FUNCTION_BLOCK FB_PistonExtruderControl EXTENDS FB_ExtruderControl

VAR
	eSubType				: E_ExtruderType;
	pFbPistonExtruderRef	: POINTER TO FB_PistonExtruderRef;
	nStateSdo 				: USINT;
	nNextStateSdo			: USINT;
	fbSdoWrite				: FB_SDO_WRITE;
	bSendDistancePending	: BOOL;
	bSendUnlockOffsetPending: BOOL;
	fbList					: FB_LinkedListCtrl;
	hList					: T_HLINKEDLIST;
	aListNodes				: ARRAY[0..6] OF T_LinkedListEntry;
	nListValue				: PVOID;
	
	bLock					: BOOL;
	nLockOffset				: DINT;
	bUnlock					: BOOL;
	nUnlockOffset			: DINT;
	bMovePlunger			: BOOL;
	nMovePos				: DINT;
	nMoveDistance			: DINT;
	nMoveFeed				: DINT;
	bExtrude				: BOOL;
	
	nCompDistanceTemp		: DINT;
	nRelaxDistanceTemp		: DINT;
	nRelaxFeedTemp			: DINT;
	nDistanceTemp			: DINT;
	nFeedTemp				: DINT;
	
	nStateAction			: USINT;
	
	timer					: TON;
	
	bStop					: BOOL;

END_VAR

VAR CONSTANT
	cMaxPosPiston	 		: DINT := 65000;//µm
	cMaxPosSyringe			: DINT := 87000;//µm
	cMaxFeedPiston			: DINT := 3000;//µm/s
	cMaxFeedSyringe			: DINT := 12000;//µm/s
END_VAR

IF pFbExtruderRef = 0 THEN
	RETURN;
END_IF

pFbPistonExtruderRef := pFbExtruderRef;

IF nStateSdo = 0 THEN //nächsten Eintrag aus Liste holen
	fbList.A_GetHead(hList:= hList,getValue=> nListValue);
	IF fbList.bOk THEN
		{IF  hasvalue (RegisterSize, '32')}
		nStateSdo := UDINT_TO_USINT(nListValue);
		{ELSE}
		nStateSdo := ULINT_TO_USINT(nListValue);
		{END_IF}		
		fbList.A_RemoveHeadValue(hList:= hList);
	END_IF
END_IF

IF nStateSdo = 1 THEN	//Feed
	fbSdoWrite(sADSNetID:= pFbPistonExtruderRef^.pMultiZRef^.P_sAdsNetId, nPortNr:= pFbPistonExtruderRef^.pMultiZRef^.P_nAdsPort, 
				nIndex:= cExtruderFeed.nIndex, nSubIndex:= pFbPistonExtruderRef^.nChannel, nDataLength:= cExtruderFeed.nLength,
				nData:= pFbPistonExtruderRef^.P_nFeedCalc, bExecute:= TRUE); 
	
ELSIF nStateSdo = 2 THEN //CompressFeed
	fbSdoWrite(sADSNetID:= pFbPistonExtruderRef^.pMultiZRef^.P_sAdsNetId, nPortNr:= pFbPistonExtruderRef^.pMultiZRef^.P_nAdsPort, 
				nIndex:= cExtruderCompressFeed.nIndex, nSubIndex:= pFbPistonExtruderRef^.nChannel, nDataLength:= cExtruderCompressFeed.nLength,
				nData:= pFbPistonExtruderRef^.P_nCompFeedCalc, bExecute:= TRUE); 
	
ELSIF nStateSdo = 3 THEN //RelaxFeed
	fbSdoWrite(sADSNetID:= pFbPistonExtruderRef^.pMultiZRef^.P_sAdsNetId, nPortNr:= pFbPistonExtruderRef^.pMultiZRef^.P_nAdsPort, 
				nIndex:= cExtruderRelaxFeed.nIndex, nSubIndex:= pFbPistonExtruderRef^.nChannel, nDataLength:= cExtruderRelaxFeed.nLength,
				nData:= pFbPistonExtruderRef^.P_nRelaxFeedCalc, bExecute:= TRUE); 
	
ELSIF nStateSdo = 4 THEN //Distance
	fbSdoWrite(sADSNetID:= pFbPistonExtruderRef^.pMultiZRef^.P_sAdsNetId, nPortNr:= pFbPistonExtruderRef^.pMultiZRef^.P_nAdsPort, 
				nIndex:= cExtruderDistance.nIndex, nSubIndex:= pFbPistonExtruderRef^.nChannel, nDataLength:= cExtruderDistance.nLength,
				nData:= pFbPistonExtruderRef^.P_nDistanceCalc, bExecute:= TRUE);
	
ELSIF nStateSdo = 5 THEN //CompressDistance
	fbSdoWrite(sADSNetID:= pFbPistonExtruderRef^.pMultiZRef^.P_sAdsNetId, nPortNr:= pFbPistonExtruderRef^.pMultiZRef^.P_nAdsPort, 
				nIndex:= cExtruderCompressDistance.nIndex, nSubIndex:= pFbPistonExtruderRef^.nChannel, nDataLength:= cExtruderCompressDistance.nLength,
				nData:= pFbPistonExtruderRef^.P_nCompDistanceCalc, bExecute:= TRUE);

ELSIF nStateSdo = 6 THEN //RelaxDistance
	fbSdoWrite(sADSNetID:= pFbPistonExtruderRef^.pMultiZRef^.P_sAdsNetId, nPortNr:= pFbPistonExtruderRef^.pMultiZRef^.P_nAdsPort, 
				nIndex:= cExtruderRelaxDistance.nIndex, nSubIndex:= pFbPistonExtruderRef^.nChannel, nDataLength:= cExtruderRelaxDistance.nLength,
				nData:= pFbPistonExtruderRef^.P_nRelaxDistanceCalc, bExecute:= TRUE);
				
ELSIF nStateSdo = 7 THEN //UnlockOffset
	fbSdoWrite(sADSNetID:= pFbPistonExtruderRef^.pMultiZRef^.P_sAdsNetId, nPortNr:= pFbPistonExtruderRef^.pMultiZRef^.P_nAdsPort, 
				nIndex:= cExtruderUnlockOffset.nIndex, nSubIndex:= pFbPistonExtruderRef^.nChannel, nDataLength:= cExtruderUnlockOffset.nLength,
				nData:= pFbPistonExtruderRef^.P_nUnlockOffsetCalc, bExecute:= TRUE);				
END_IF

IF NOT fbSdoWrite.bBusy THEN
	IF fbSdoWrite.bError THEN
		bError := TRUE;
		nErrorId := fbSdoWrite.nAdsErrorId;		
	END_IF
	fbSdoWrite(bExecute:= FALSE);
	IF nStateSdo = 4 THEN
		bSendDistancePending := FALSE;
	ELSIF nStateSdo = 7 THEN
		bSendUnlockOffsetPending := FALSE;
	END_IF
	nStateSdo := 0;
END_IF


IF bLock THEN
	A_Lock();
ELSIF bUnlock THEN
	A_Unlock();
ELSIF bMovePlunger THEN
	A_MovePlunger();
ELSIF bExtrude THEN
	A_Extrude();
END_IF

IF nStateAction >= 80 THEN
	IF nStateAction >= 99 THEN
		bError := TRUE;
	END_IF
	bLock := bUnlock := bMovePlunger := bExtrude := FALSE;
	nStateAction := 0;
END_IF

bBusy := bLock OR bUnlock OR bMovePlunger OR bExtrude;

ACTION A_Extrude:
CASE nStateAction OF
	0:	//warten, bis Distance gesendet
		IF NOT bSendDistancePending THEN
			pFbPistonExtruderRef^.pToolCtrl^.0 := TRUE;
			nStateAction := 1;				
		END_IF
		
	1:	//Timeout für active
		timer(IN:=TRUE,PT:=T#1S);
		IF pFbPistonExtruderRef^.P_bIsActive THEN
			timer(IN:=FALSE);
			nStateAction := 2;
		ELSE
			IF timer.Q THEN
				timer(IN:=FALSE);
				nErrorId := E_ErrorIdMultiZ.ERRORID_TimeoutExtrude;
				pFbPistonExtruderRef^.pToolCtrl^ := 0;
				nStateAction := 99;
			END_IF
		END_IF
		
	2:	//warten, bis Extrude fertig
		IF NOT pFbPistonExtruderRef^.P_bIsActive OR bStop THEN
			bStop := FALSE;
			pFbPistonExtruderRef^.pToolCtrl^.0 := FALSE;
			nStateAction := 80;
		END_IF
	
END_CASE
END_ACTION

ACTION A_Lock:
CASE nStateAction OF
	0:	//Wartezyklus
		IF pFbPistonExtruderRef^.P_bIsActive THEN
			nStateAction := 99;
		ELSE
			nStateAction := 1;
		END_IF
	1:	//Locking starten
		pFbPistonExtruderRef^.pToolCtrl^.0 := TRUE;
		pFbPistonExtruderRef^.pToolCtrl^.2 := TRUE;
		//Timeout für active
		timer(IN:=TRUE,PT:=T#1S);
		IF pFbPistonExtruderRef^.P_bIsActive THEN
			pFbPistonExtruderRef^.pToolCtrl^.0 := FALSE;
			timer(IN:=FALSE);
			nStateAction := 2;
		ELSE
			IF timer.Q THEN
				timer(IN:=FALSE);
				nErrorId := E_ErrorIdMultiZ.ERRORID_TimeoutLock;
				nStateAction := 99;
			END_IF
		END_IF
		
	2:	//waiting for "ready state"
		timer(IN:=TRUE,PT:=T#25S);
		IF NOT pFbPistonExtruderRef^.P_bIsActive THEN
			timer(IN:=FALSE);
			IF nLockOffset > 0 AND NOT pFbPistonExtruderRef^.pToolCtrl^.1 THEN
				nStateAction := 3;
			ELSE
				nStateAction := 80;
			END_IF
			pFbPistonExtruderRef^.pToolCtrl^ := 0;
		ELSE
			IF timer.Q THEN
				timer(IN:=FALSE);
				nErrorId := E_ErrorIdMultiZ.ERRORID_TimeoutLock;
				nStateAction := 99;
			END_IF
		END_IF
		
	3:	//auf Offset fahren
		//aktuelle CompDistance, RelaxDistance, Feed, Distance sichern
		nCompDistanceTemp := pFbPistonExtruderRef^.P_nCompDistanceOrgin;
		nRelaxDistanceTemp := pFbPistonExtruderRef^.P_nRelaxDistanceOrgin;
		nFeedTemp := pFbPistonExtruderRef^.P_nFeedOrgin;
		nDistanceTemp := pFbPistonExtruderRef^.P_nDistanceOrgin;
		
		//CompDist + RelaxDist auf 0 setzen
		M_SetCompDistance(0);
		M_SetRelaxDistance(0);
		nMoveFeed := M_SetFeedToMax();
		M_SetDistance(nLockOffset); //Distance auf Offset setzen
		nStateAction := 4;
		
	4:	//warten bis Distance gesendet (andere werden vorher gesendet)
		IF NOT bSendDistancePending THEN
			pFbPistonExtruderRef^.pToolCtrl^.0 := TRUE;
			timer(IN:=FALSE);
			nStateAction := 5;
		END_IF
		
	5:	//waiting for "active state"
		timer(IN:=TRUE,PT:=T#1S);
		IF pFbPistonExtruderRef^.P_bIsActive THEN
			timer(IN:=FALSE);
			//timeout berechnen
			timer.PT := REAL_TO_TIME((DINT_TO_REAL(nLockOffset) / DINT_TO_REAL(nMoveFeed))*10000.0 + 3000.0);
			nStateAction := 6;
		ELSE
			IF timer.Q THEN
				timer(IN:=FALSE);
				nErrorId := E_ErrorIdMultiZ.ERRORID_TimeoutLock;
				nStateAction := 7;
			END_IF
		END_IF
		
	6:	//waiting for "ready state"
		timer(IN:=TRUE);
		IF NOT pFbPistonExtruderRef^.P_bIsActive THEN
			timer(IN:=FALSE);
			pFbPistonExtruderRef^.pToolCtrl^ := 0;
			nStateAction := 7;
		ELSE
			IF timer.Q THEN
				timer(IN:=FALSE);
				nErrorId := E_ErrorIdMultiZ.ERRORID_TimeoutLock;
				nStateAction := 7;
			END_IF
		END_IF
		
	7:	//gesicherte Parameter zurückschreiben
		M_SetCompDistance(nCompDistanceTemp);
		M_SetRelaxDistance(nRelaxDistanceTemp);
		M_SetFeed(nFeedTemp);
		M_SetDistance(nDistanceTemp);
		nStateAction := 8;

	8:	//warten bis Distance gesendet (andere werden vorher gesendet)
		IF NOT bSendDistancePending THEN
			IF nErrorId > 0 THEN
				nStateAction := 99;
			ELSE
				nStateAction := 80;
			END_IF
		END_IF		

END_CASE

IF nStateAction = 99 THEN
	pFbPistonExtruderRef^.pToolCtrl^ := 0;
END_IF
END_ACTION

ACTION A_MovePlunger:
//Ähnlich wie Extrude impl.
//vorher aktuelle Position von Zielposition abziehen
//CompDist und RelaxDist auf 0 setzen
CASE nStateAction OF
	0:	//aktuelle CompDistance, RelaxDistance, Feed, Distance sichern
		nCompDistanceTemp := pFbPistonExtruderRef^.P_nCompDistanceOrgin;
		nRelaxDistanceTemp := pFbPistonExtruderRef^.P_nRelaxDistanceOrgin;
		nRelaxFeedTemp := pFbPistonExtruderRef^.P_nRelaxFeedOrgin;
		nFeedTemp := pFbPistonExtruderRef^.P_nFeedOrgin;
		nDistanceTemp := pFbPistonExtruderRef^.P_nDistanceOrgin;
		
		nStateAction := 1;

		M_SetCompDistance(0);
		IF nMovePos > pFbPistonExtruderRef^.P_nCurrentPos THEN
			M_SetRelaxDistance(0);
			nMoveFeed := M_SetFeedToMax();
			nMoveDistance := nMovePos - pFbPistonExtruderRef^.P_nCurrentPos; 
			M_SetDistance(nMoveDistance);
		ELSIF nMovePos < pFbPistonExtruderRef^.P_nCurrentPos THEN
			nMoveDistance := pFbPistonExtruderRef^.P_nCurrentPos - nMovePos;
			M_SetRelaxDistance(nMoveDistance);
			nMoveFeed := M_SetRelaxFeedToMax();
			M_SetFeedToMax();
			M_SetDistance(1);
		ELSE
			nStateAction := 80;
			RETURN;
		END_IF
		
	1:	//warten bis Distance gesendet (andere werden vorher gesendet)
		IF NOT bSendDistancePending THEN
			pFbPistonExtruderRef^.pToolCtrl^.0 := TRUE;
			nStateAction := 2;
		END_IF
		
	2:	//waiting for "active state"
		timer(IN:=TRUE,PT:=T#1S);
		IF pFbPistonExtruderRef^.P_bIsActive THEN
			timer(IN:=FALSE);
			//timeout berechnen
			timer.PT := REAL_TO_TIME((DINT_TO_REAL(nMoveDistance) / DINT_TO_REAL(nMoveFeed))*10000.0 + 3000.0);
			nStateAction := 3;
		ELSE
			IF timer.Q THEN
				timer(IN:=FALSE);
				nErrorId := E_ErrorIdMultiZ.ERRORID_TimeoutMovePlunger;
				nStateAction := 4;
			END_IF
		END_IF	
		
	3:	//warten, bis Extrude fertig
		timer(IN:=TRUE);
		IF NOT pFbPistonExtruderRef^.P_bIsActive THEN
			timer(IN:=FALSE);
			pFbPistonExtruderRef^.pToolCtrl^ := 0;
			nStateAction := 4;
		ELSE
			IF timer.Q THEN
				timer(IN:=FALSE);
				nErrorId := E_ErrorIdMultiZ.ERRORID_TimeoutMovePlunger;
				nStateAction := 4;
			END_IF
		END_IF
		
	4:	//gesicherte Parameter zurückschreiben
		M_SetCompDistance(nCompDistanceTemp);
		M_SetRelaxDistance(nRelaxDistanceTemp);
		M_SetRelaxFeed(nRelaxFeedTemp);
		M_SetFeed(nFeedTemp);
		M_SetDistance(nDistanceTemp);
		nStateAction := 5;
		
	5:	//warten bis Distance gesendet (andere werden vorher gesendet)
		IF NOT bSendDistancePending THEN
			IF nErrorId > 0 THEN
				nStateAction := 99;
			ELSE
				nStateAction := 80;	
			END_IF
		END_IF			
END_CASE

IF nStateAction = 99 THEN
	pFbPistonExtruderRef^.pToolCtrl^ := 0;
END_IF
END_ACTION

ACTION A_Unlock:
CASE nStateAction OF
	0:	//warten bis nUnlockOffset übertragen
		IF NOT bSendUnlockOffsetPending THEN
			nStateAction := 1;
		END_IF
		
	1:	//UnLocking starten
		pFbPistonExtruderRef^.pToolCtrl^.0 := TRUE;
		pFbPistonExtruderRef^.pToolCtrl^.2 := TRUE;
		//Timeout für active
		timer(IN:=TRUE,PT:=T#1S);
		IF pFbPistonExtruderRef^.P_bIsActive THEN
			pFbPistonExtruderRef^.pToolCtrl^.0 := FALSE;
			timer(IN:=FALSE);
			nStateAction := 2;
		ELSE
			IF timer.Q THEN
				timer(IN:=FALSE);
				nErrorId := E_ErrorIdMultiZ.ERRORID_TimeoutUnLock;
				nStateAction := 99;
			END_IF
		END_IF
		
	2:	//warten, bis UnLocking ready
		timer(IN:=TRUE,PT:=T#70S);
		IF NOT pFbPistonExtruderRef^.P_bIsActive THEN
			timer(IN:=FALSE);
			pFbPistonExtruderRef^.pToolCtrl^ := 0;
			nStateAction := 80;
		ELSE
			IF timer.Q THEN
				timer(IN:=FALSE);
				nErrorId := E_ErrorIdMultiZ.ERRORID_TimeoutUnLock;
				nStateAction := 99;
			END_IF
		END_IF
END_CASE

IF nStateAction = 99 THEN
	pFbPistonExtruderRef^.pToolCtrl^ := 0;
END_IF
END_ACTION

METHOD FB_init : BOOL
VAR_INPUT
	bInitRetains : BOOL; // if TRUE, the retain variables are initialized (warm start / cold start)
	bInCopyCode : BOOL;  // if TRUE, the instance afterwards gets moved into the copy code (online change)
END_VAR
F_CreateLinkedListHnd(ADR(aListNodes ), SIZEOF(aListNodes ), hList);
END_METHOD

METHOD PRIVATE M_Add
VAR_INPUT
	nValue : UDINT;
END_VAR
VAR
	pPosPtr	: POINTER TO T_LinkedListEntry := 0;
END_VAR
//Checken, ob Eintrag schon vorhanden
fbList.A_GetHead(hList:= hList,getValue=> nListValue, getPosPtr=> pPosPtr);
IF fbList.bOk THEN
	IF nValue = nListValue THEN	//Eintrag schon vorhanden
		RETURN;		
	ELSE //Eintrag nicht vorhanden -> weitersuchen
		REPEAT
			fbList.A_GetNext(hList:= hList,getValue=> nListValue, putPosPtr:= pPosPtr, getPosPtr=> pPosPtr);
			IF fbList.bOk THEN
				IF nValue = nListValue THEN	//Eintrag schon vorhanden
					RETURN;
				END_IF
			END_IF
		UNTIL NOT fbList.bOk
		END_REPEAT
	END_IF
END_IF

fbList.A_AddTailValue(hList:= hList, putValue:= nValue);
END_METHOD

METHOD M_HardStop
VAR_INPUT
END_VAR
IF pFbPistonExtruderRef^.P_bIsActive THEN
	pFbPistonExtruderRef^.pToolCtrl^ := 2;
END_IF
END_METHOD

METHOD M_Init
VAR_INPUT
END_VAR

VAR
	i : USINT;
END_VAR
//Alle Parameter übertragen
FOR i := 1 TO 7 BY 1 DO
	M_Add(i);
END_FOR
END_METHOD

METHOD M_Lock
VAR_INPUT
	nOffset : DINT;
END_VAR
IF NOT (pFbPistonExtruderRef^.P_bIsActive OR pFbExtruderRef^.P_bError OR bBusy) THEN
	nLockOffset := nOffset;
	pFbPistonExtruderRef^.pToolCtrl^ := 0;
	bBusy := TRUE;
	bLock := TRUE;	
END_IF
END_METHOD

METHOD M_MovePlunger
VAR_INPUT
	nPosition : DINT;
END_VAR
nMovePos := nPosition;
IF  NOT(pFbPistonExtruderRef^.P_bIsActive OR pFbPistonExtruderRef^.P_bError OR bBusy) THEN
	bBusy := TRUE;
	bMovePlunger := TRUE;
	pFbPistonExtruderRef^.pToolCtrl^ := 0;
END_IF
END_METHOD

METHOD M_SetCompDistance : ERRORID
VAR_INPUT
		nValue : DINT;
END_VAR

VAR
	nMaxCompPos : DINT;
END_VAR
IF eSubType = E_ExtruderType.PistonExtruder1 THEN
	nMaxCompPos  := cMaxPosPiston;
ELSIF eSubType = E_ExtruderType.SyringeExtruder1 THEN
	nMaxCompPos  := cMaxPosSyringe;
ELSE
	M_SetCompDistance := E_ErrorIdObjMgmt.ERRORID_InvalidExtruderSubType;
END_IF

IF nValue >= 0 AND nValue <= nMaxCompPos THEN
	IF pFbPistonExtruderRef > 0 THEN
		IF pFbPistonExtruderRef^.P_nCompDistanceOrgin <> nValue THEN
			pFbPistonExtruderRef^.P_nCompDistanceOrgin := nValue;
			M_Add(5);
		END_IF
	END_IF
ELSE
	M_SetCompDistance := E_ErrorIdObjMgmt.ERRORID_InvalidCompressDistance;
END_IF
END_METHOD

METHOD M_SetCompFeed : ERRORID
VAR_INPUT
	nValue : DINT;
END_VAR

VAR
	nMaxCompFeed : DINT;
END_VAR
IF eSubType = E_ExtruderType.PistonExtruder1 THEN
	nMaxCompFeed := cMaxFeedPiston;
ELSIF eSubType = E_ExtruderType.SyringeExtruder1 THEN
	nMaxCompFeed := cMaxFeedSyringe;
ELSE
	M_SetCompFeed := E_ErrorIdObjMgmt.ERRORID_InvalidExtruderSubType;
END_IF

IF nValue >= 0 AND nValue <= nMaxCompFeed THEN
	IF pFbPistonExtruderRef > 0 THEN
		IF pFbPistonExtruderRef^.P_nCompFeedOrgin <> nValue THEN
			pFbPistonExtruderRef^.P_nCompFeedOrgin := nValue;
			M_Add(2);
		END_IF
	END_IF
ELSE
	M_SetCompFeed := E_ErrorIdObjMgmt.ERRORID_InvalidCompressFeed;
END_IF
END_METHOD

METHOD M_SetDistance : ERRORID
VAR_INPUT
	nValue : DINT;
END_VAR

VAR
	nMaxPos : DINT;
END_VAR
IF eSubType = E_ExtruderType.PistonExtruder1 THEN
	nMaxPos := cMaxPosPiston;
ELSIF eSubType = E_ExtruderType.SyringeExtruder1 THEN
	nMaxPos := cMaxPosSyringe;
ELSE
	M_SetDistance := E_ErrorIdObjMgmt.ERRORID_InvalidExtruderSubType;
END_IF

IF nValue >= 0 AND nValue <= nMaxPos THEN
	IF pFbPistonExtruderRef > 0 THEN
		IF pFbPistonExtruderRef^.P_nDistanceOrgin <> nValue THEN
			pFbPistonExtruderRef^.P_nDistanceOrgin := nValue;
			M_Add(4);
			bSendDistancePending := TRUE;
		END_IF
	END_IF
ELSE
	M_SetDistance := E_ErrorIdObjMgmt.ERRORID_InvalidExtrudeDistance;
END_IF
END_METHOD

METHOD M_SetFeed : ERRORID
VAR_INPUT
	nValue : DINT;
END_VAR

VAR
	nMaxFeed : DINT;
END_VAR
IF eSubType = E_ExtruderType.PistonExtruder1 THEN
	nMaxFeed := cMaxFeedPiston;
ELSIF eSubType = E_ExtruderType.SyringeExtruder1 THEN
	nMaxFeed := cMaxFeedSyringe;
ELSE
	M_SetFeed := E_ErrorIdObjMgmt.ERRORID_InvalidExtruderSubType;
END_IF

IF nValue >= 0 AND nValue <= nMaxFeed THEN
	IF pFbPistonExtruderRef > 0 THEN
		IF pFbPistonExtruderRef^.P_nFeedOrgin <> nValue THEN
			pFbPistonExtruderRef^.P_nFeedOrgin := nValue;
			M_Add(1);
		END_IF
	END_IF
ELSE
	M_SetFeed := E_ErrorIdObjMgmt.ERRORID_InvalidExtrudeFeed;
END_IF
END_METHOD

METHOD M_SetFeedToMax : DINT
VAR_INPUT
END_VAR
IF eSubType = E_ExtruderType.PistonExtruder1 THEN
	M_SetFeed(cMaxFeedPiston);
	M_SetFeedToMax := cMaxFeedPiston;
ELSIF eSubType = E_ExtruderType.SyringeExtruder1 THEN
	M_SetFeed(cMaxFeedSyringe);
	M_SetFeedToMax := cMaxFeedSyringe;
END_IF
END_METHOD

METHOD M_SetRelaxDistance : ERRORID
VAR_INPUT
	nValue : DINT;
END_VAR

VAR
	nMaxRelaxPos : DINT;
END_VAR
IF eSubType = E_ExtruderType.PistonExtruder1 THEN
	nMaxRelaxPos := cMaxPosPiston;
ELSIF eSubType = E_ExtruderType.SyringeExtruder1 THEN
	nMaxRelaxPos := cMaxPosSyringe;
ELSE
	M_SetRelaxDistance := E_ErrorIdObjMgmt.ERRORID_InvalidExtruderSubType;
END_IF

IF nValue >= 0 AND nValue <= nMaxRelaxPos THEN
	IF pFbPistonExtruderRef > 0 THEN
		IF pFbPistonExtruderRef^.P_nRelaxDistanceOrgin <> nValue THEN
			pFbPistonExtruderRef^.P_nRelaxDistanceOrgin := nValue;
			M_Add(6);
		END_IF
	END_IF
ELSE
	M_SetRelaxDistance := E_ErrorIdObjMgmt.ERRORID_InvalidRelaxDistance;
END_IF
END_METHOD

METHOD M_SetRelaxFeed : ERRORID
VAR_INPUT
	nValue : DINT;
END_VAR

VAR
	nMaxRelaxFeed : DINT;
END_VAR
IF eSubType = E_ExtruderType.PistonExtruder1 THEN
	nMaxRelaxFeed := cMaxFeedPiston;
ELSIF eSubType = E_ExtruderType.SyringeExtruder1 THEN
	nMaxRelaxFeed := cMaxFeedSyringe;
ELSE
	M_SetRelaxFeed := E_ErrorIdObjMgmt.ERRORID_InvalidExtruderSubType;
END_IF

IF nValue >= 0 AND nValue <= nMaxRelaxFeed THEN
	IF pFbPistonExtruderRef > 0 THEN
		IF pFbPistonExtruderRef^.P_nRelaxFeedOrgin <> nValue THEN
			pFbPistonExtruderRef^.P_nRelaxFeedOrgin := nValue;
			M_Add(3);
		END_IF
	END_IF
ELSE
	M_SetRelaxFeed := E_ErrorIdObjMgmt.ERRORID_InvalidRelaxFeed;	
END_IF
END_METHOD

METHOD M_SetRelaxFeedToMax : DINT
VAR_INPUT
END_VAR
IF eSubType = E_ExtruderType.PistonExtruder1 THEN
	M_SetRelaxFeed(cMaxFeedPiston);
	M_SetRelaxFeedToMax := cMaxFeedPiston;
ELSIF eSubType = E_ExtruderType.SyringeExtruder1 THEN
	M_SetRelaxFeed(cMaxFeedSyringe);
	M_SetRelaxFeedToMax := cMaxFeedSyringe;
END_IF
END_METHOD

METHOD M_SetUnlockOffset : ERRORID
VAR_INPUT
	nValue : DINT;
END_VAR

VAR
	nMaxUnlockOffset : DINT;
END_VAR
IF eSubType = E_ExtruderType.PistonExtruder1 THEN
	nMaxUnlockOffset := cMaxPosPiston;
ELSIF eSubType = E_ExtruderType.SyringeExtruder1 THEN
	nMaxUnlockOffset := cMaxPosSyringe;
ELSE
	M_SetUnlockOffset := E_ErrorIdObjMgmt.ERRORID_InvalidExtruderSubType;
END_IF

IF nValue >= 0 AND nValue <= nMaxUnlockOffset THEN
	IF pFbPistonExtruderRef > 0 THEN
		IF pFbPistonExtruderRef^.P_nUnlockOffsetOrgin <> nValue THEN
			pFbPistonExtruderRef^.P_nUnlockOffsetOrgin := nValue;
			M_Add(7);
			bSendUnlockOffsetPending := TRUE;
		END_IF
	END_IF
ELSE
	M_SetUnlockOffset := E_ErrorIdObjMgmt.ERRORID_InvalidUnlockOffset;	
END_IF
END_METHOD

METHOD M_StartStop
VAR_INPUT
	bStart : BOOL;
END_VAR
//Extruder darf nur gestartet werden, wenn:
//1. Das Status-bit ist nicht gesetzt
//2. er ist nicht in Error

IF bStart AND NOT (pFbPistonExtruderRef^.P_bIsActive OR pFbPistonExtruderRef^.P_bError OR bBusy) THEN
	bBusy := TRUE;
	bExtrude := TRUE;
	bStop := FALSE;
	pFbPistonExtruderRef^.pToolCtrl^.1 := FALSE; //HardStop
	pFbPistonExtruderRef^.pToolCtrl^.2 := FALSE; //Mode "Lock/Unlock"
ELSE
	bStop := TRUE;
END_IF
END_METHOD

METHOD M_Unlock
VAR_INPUT
	nOffset : DINT;
END_VAR
IF NOT (pFbPistonExtruderRef^.P_bIsActive OR pFbExtruderRef^.P_bError OR bBusy) THEN
	nUnlockOffset := nOffset;
	M_SetUnlockOffset(nUnlockOffset);
	pFbPistonExtruderRef^.pToolCtrl^.2 := FALSE;
	bBusy := TRUE;
	bUnLock := TRUE;
END_IF
END_METHOD

PROPERTY P_eSubType : E_ExtruderType
GET
P_eSubType := eSubType;
END_GET
SET
eSubType := P_eSubType;
END_SET
END_PROPERTY

PROPERTY P_nMaxPos : DINT
GET
IF eSubType = E_ExtruderType.PistonExtruder1 THEN
	P_nMaxPos := cMaxPosPiston;
ELSIF eSubType = E_ExtruderType.SyringeExtruder1 THEN
	P_nMaxPos := cMaxPosSyringe;
END_IF
END_GET
END_PROPERTY

END_FUNCTION_BLOCK

(* stored: Version 1.1.0.1, ProductVersion 3.1.4022.18
   POU FB_PistonExtruderControl: Id {e81a9316-202c-4324-8f9c-757019bef4b3}, SpecialFunc None
   Action A_Extrude: Id {cbbeb795-f017-486a-a146-c756f9c8af36}
   Action A_Lock: Id {fc30b96a-fc15-449c-8aad-3a49d43240a8}
   Action A_MovePlunger: Id {52873978-f7b4-4179-85d8-663bea95e237}
   Action A_Unlock: Id {a98f7662-7402-4d8b-aaed-e9a256bae2f3}
   Method FB_init: Id {ad08ff75-f75f-4d4e-899b-a26246863797}
   Method M_Add: Id {12b0027a-0213-46a0-bee7-338ff0559525}
   Method M_HardStop: Id {cf72ab57-c2e2-4b83-99a9-25c7f9c24e9e}
   Method M_Init: Id {dce0e30f-6c7c-4159-9792-3884a0fde4dd}
   Method M_Lock: Id {7420e009-b527-44b6-9232-21b3000a9ced}
   Method M_MovePlunger: Id {38e60e70-e6a5-4b52-a900-86710b6fc9f2}
   Method M_SetCompDistance: Id {f27db045-b279-43ed-a422-eae536a4a5a8}
   Method M_SetCompFeed: Id {af54794a-3074-406e-a512-ebf846531dfd}
   Method M_SetDistance: Id {34b4b23e-096a-48d3-8ddf-55c6dee1e3ca}
   Method M_SetFeed: Id {839d52e2-6609-482f-816c-1649a2130ac9}
   Method M_SetFeedToMax: Id {7644cab0-bcfb-4d8b-8c71-e7e1e5ba5222}
   Method M_SetRelaxDistance: Id {8ebd5eb2-be1c-498f-85fd-680e3e284565}
   Method M_SetRelaxFeed: Id {30677a91-e6ba-474e-abd8-7aa0b7a14a33}
   Method M_SetRelaxFeedToMax: Id {01a14a88-5ca4-431d-8c5e-f5fc04731720}
   Method M_SetUnlockOffset: Id {4dccb08a-18ea-4482-9435-0f85dd43bcee}
   Method M_StartStop: Id {a7d55010-a248-4e87-b7d9-dd3617b51ee5}
   Method M_Unlock: Id {cc8bb752-49e5-491c-86f9-29c8e3cc5498}
   Property P_eSubType: Id {992420da-7e6f-4629-a2f1-0876edbe31a9}
   Get Get: Id {69605781-ddd0-45c9-989e-89d5e51a07d1}
   Set Set: Id {c004b309-5d0c-4b33-858e-5baf5b4d4f0f}
   Property P_nMaxPos: Id {3c095b0e-bd84-4c83-ba07-7049027e6496}
   Get Get: Id {2e9de394-19d0-48a1-9af7-5ec5b9c1fe64} *)
